{attribute 'no_explicit_call' := 'do not call this function block directly'} 
FUNCTION_BLOCK FileContentManager EXTENDS ToolkitObject IMPLEMENTS IAbortableProcess
VAR
	_ClassName : STRING := __POUNAME();

	_FilePath : Tc2_System.T_MaxString;	
	_OpenMode : FILE_OPEN_MODE;
	_ContentHandlingMode : FILE_CONTENT_HANDLING_MODE;
	_PathType : E_OpenPath;	
	_AmsNetId : Tc2_System.T_AmsNetID;
	_FileHandle : UINT;
		
	_TaskExecutor : SequentialTaskExecutor;
END_VAR

{attribute 'monitoring' := 'call'}
{attribute 'OPC.UA.DA.Property' := '1'}
{attribute 'OPC.UA.DA.Access' := '1'}
PROPERTY FINAL Aborted : BOOL
GET
Aborted := _TaskExecutor.Aborted;
END_GET
END_PROPERTY

{attribute 'monitoring' := 'call'}
{attribute 'OPC.UA.DA.Property' := '1'}
{attribute 'OPC.UA.DA.Access' := '1'}
PROPERTY FINAL Aborting : BOOL
GET
Busy := _TaskExecutor.Busy;
END_GET
END_PROPERTY

{attribute 'monitoring' := 'call'}
{attribute 'OPC.UA.DA.Property' := '1'}
{attribute 'OPC.UA.DA.Access' := '1'}
PROPERTY AbortReason : REFERENCE TO ERROR_MESSAGE
GET
AbortReason REF= _TaskExecutor.AbortReason;
END_GET
END_PROPERTY

METHOD AddTask
VAR_INPUT
	fileOperation : REFERENCE TO FileContentTask;
END_VAR
IF __ISVALIDREF(fileOperation) THEN
	fileOperation.FileContentManager REF= THIS^;

	_TaskExecutor.AddTask(fileOperation);
END_IF
END_METHOD

{attribute 'monitoring' := 'call'}
{attribute 'OPC.UA.DA.Property' := '1'}
PROPERTY AmsNetId : Tc2_System.T_AmsNetID
GET
AmsNetId := _AmsNetId;
END_GET
SET
_AmsNetId := AmsNetId;
END_SET
END_PROPERTY

{attribute 'monitoring' := 'call'}
{attribute 'OPC.UA.DA.Property' := '1'}
{attribute 'OPC.UA.DA.Access' := '1'}
PROPERTY FINAL Busy : BOOL
GET
Busy := _TaskExecutor.Busy;
END_GET
END_PROPERTY

{attribute 'monitoring' := 'call'}
PROPERTY ClassName : STRING
GET
ClassName := _ClassName;
END_GET
END_PROPERTY

{attribute 'monitoring' := 'call'}
{attribute 'OPC.UA.DA.Property' := '1'}
{attribute 'OPC.UA.DA.Access' := '1'}
PROPERTY ContentHandlingMode : FILE_CONTENT_HANDLING_MODE
GET
ContentHandlingMode := _ContentHandlingMode;
END_GET
SET // INTERNAL
_ContentHandlingMode := ContentHandlingMode;
END_SET
END_PROPERTY

{attribute 'monitoring' := 'call'}
{attribute 'OPC.UA.DA.Property' := '1'}
{attribute 'OPC.UA.DA.Access' := '1'}
PROPERTY FINAL Error : BOOL
GET
Error := _TaskExecutor.Error;
END_GET
END_PROPERTY

{attribute 'monitoring' := 'call'}
{attribute 'OPC.UA.DA.Property' := '1'}
{attribute 'OPC.UA.DA.Access' := '1'}
PROPERTY FINAL ErrorMessage : REFERENCE TO Exception
GET
ErrorMessage REF= _TaskExecutor.ErrorMessage;
END_GET
END_PROPERTY

METHOD Execute
_TaskExecutor.Execute();
END_METHOD

METHOD FB_exit : BOOL
VAR_INPUT
	bInCopyCode : BOOL; // if TRUE, the exit method is called for exiting an instance that is copied afterwards (online change).
END_VAR
VAR_INST
	_Close : Tc2_System.FB_FileClose;
END_VAR
IF _FileHandle <> 0 THEN
	_Close(
		bExecute := TRUE,
		hFile := _FileHandle,
		sNetId := _AmsNetId,
		tTimeout := T#1S		
	); 
END_IF
END_METHOD

METHOD FB_init : BOOL
VAR_INPUT
	bInitRetains : BOOL; // if TRUE, the retain variables are initialized (warm start / cold start)
	bInCopyCode : BOOL; // if TRUE, the instance afterwards gets moved into the copy code (online change)
END_VAR
_TaskExecutor.ContinueOnTaskError := TRUE;
END_METHOD

PROPERTY FileHandle : UINT
GET
FileHandle := _FileHandle;
END_GET
SET // INTERNAL
_FileHandle := FileHandle;
END_SET
END_PROPERTY

{attribute 'monitoring' := 'call'}
{attribute 'OPC.UA.DA.Property' := '1'}
{attribute 'OPC.UA.DA.Access' := '1'}
PROPERTY FilePath : Tc2_System.T_MaxString
GET
FilePath := _FilePath;
END_GET
SET // INTERNAL
_FilePath := FilePath;
END_SET
END_PROPERTY

{attribute 'monitoring' := 'call'}
{attribute 'OPC.UA.DA.Property' := '1'}
{attribute 'OPC.UA.DA.Access' := '1'}
PROPERTY IsOpen : BOOL
GET
IsOpen := _FileHandle <> 0;
END_GET
END_PROPERTY

{attribute 'monitoring' := 'call'}
{attribute 'OPC.UA.DA.Property' := '1'}
{attribute 'OPC.UA.DA.Access' := '1'}
PROPERTY OpenMode : FILE_OPEN_MODE
GET
OpenMode := _OpenMode;
END_GET
SET // INTERNAL
_OpenMode := OpenMode;
END_SET
END_PROPERTY

{attribute 'monitoring' := 'call'}
{attribute 'OPC.UA.DA.Property' := '1'}
{attribute 'OPC.UA.DA.Access' := '1'}
PROPERTY PathType : E_OpenPath
GET
PathType := _PathType;
END_GET
SET // INTERNAL
_PathType := PathType;
END_SET
END_PROPERTY

METHOD RequestAbort
VAR_INPUT 
	reason : ERROR_MESSAGE;
END_VAR
_TaskExecutor.RequestAbort(reason);
END_METHOD

METHOD Start
_TaskExecutor.Start();
END_METHOD

END_FUNCTION_BLOCK

(* stored: Version 1.1.0.1
   POU FileContentManager: Id {fdc9580e-5ae4-4706-b8f8-0dfdf87f7bef}, SpecialFunc None
   Property Aborted: Id {9e3df4ea-b68a-4946-8dd2-2ca42cbdd1a0}
   Get Get: Id {68845d3e-c6e8-4b12-8686-310e9ae7ed22}
   Property Aborting: Id {1b0ac3e4-64ba-43db-9f3c-746a7991fda2}
   Get Get: Id {63a036d1-0566-45b7-bfa5-f88f84270111}
   Property AbortReason: Id {814ebd23-7b40-4189-941d-52e79827bf77}
   Get Get: Id {117cc237-fb3f-4560-9263-0bcb57e314e0}
   Method AddTask: Id {383660f1-5947-48c8-94de-1c4ef4024d44}
   Property AmsNetId: Id {6888dca5-b51a-411f-b793-ee68602b138a}
   Get Get: Id {51d3526c-efc7-418e-9925-4e62484508ab}
   Set Set: Id {9a8f2703-9299-489b-90cf-a033342d716d}
   Property Busy: Id {7bf66eba-51f2-433a-b8d5-3a87522a7d72}
   Get Get: Id {4792156b-26bf-43b9-b714-87a5a91ac0bc}
   Property ClassName: Id {76cdd9f1-1152-49b5-9ae0-5be443d931d1}
   Get Get: Id {3ade8b3b-8429-49d3-8225-bff27db26bd1}
   Property ContentHandlingMode: Id {d775deba-40f9-49fc-b5d0-6123d2ea1175}
   Get Get: Id {e516c938-b048-41c5-82e9-4fa763e92a13}
   Set Set: Id {9705fe2c-a6d3-476e-944a-00279379a5e5}
   Property Error: Id {5f7eaf79-653e-4992-bf07-c4f353526447}
   Get Get: Id {47fb1aab-ac8c-4ed4-8fb3-820120a681e3}
   Property ErrorMessage: Id {27e40ad8-87c5-4314-a637-45e42df85154}
   Get Get: Id {f97b2d95-d4d9-40a8-8be7-3ac4e2de4116}
   Method Execute: Id {9162ff2d-545b-457a-978b-d136442fb0f6}
   Method FB_exit: Id {c22df983-6350-47b5-8a38-ffdd2fb1d664}
   Method FB_init: Id {8526a5c8-d491-432e-99d1-80424758a8b4}
   Property FileHandle: Id {dc3ea81e-f9c4-4fe9-b571-208da3ecce3b}
   Get Get: Id {cb6cfff2-2892-441b-9a24-f3c2668b0a99}
   Set Set: Id {c65f3bce-1749-478b-bcf6-9ae22053a439}
   Property FilePath: Id {fb101c5b-d564-436a-8959-480be1d5196d}
   Get Get: Id {7d4603c3-8b55-41c6-827d-871d0c3bea3d}
   Set Set: Id {a3c99c27-c24d-4fdb-8e38-9eafd21795f0}
   Property IsOpen: Id {7f658d02-4e4e-4294-ac5a-4983fd8071ce}
   Get Get: Id {896333da-d22b-4e67-9e3c-7f856f776342}
   Property OpenMode: Id {d5d409ce-c7ba-4b4b-a898-8f19d2527f17}
   Get Get: Id {f7bdcbaa-d2fc-4ef8-9a57-ca0bd077c894}
   Set Set: Id {e0c3987e-0c7b-438c-a9fa-24bc8eb121aa}
   Property PathType: Id {0ddf8fcf-9f1f-4f51-8a18-553cc072f295}
   Get Get: Id {9c387b83-683b-40dc-8d96-516089809632}
   Set Set: Id {207748d8-6f8e-40bf-b6a1-19cfb6eaea27}
   Method RequestAbort: Id {9a3d703c-ceda-4338-9739-2beeced490eb}
   Method Start: Id {5bcb3f72-0958-470f-b997-87f391014695} *)
